(* Verify that the statuses of the switchbox pumps match the expected statuses *)
FUNCTION F_VerifySBPumpStatuses : BOOL
VAR_INPUT
	stExpStatus : ST_SBPumpStatuses; // The expected state of the system
	bEnforce : BOOL; // Whether to try forcing the states
END_VAR
VAR
	stStatus : ST_SBPumpStatuses;
END_VAR

stStatus := F_GetSBPumpStatuses();

IF bEnforce THEN
	// Try setting system states to the expected states
	F_SetSBPumpStatuses(stExpStatus);
END_IF

// Return true if the expected status matches the actual status
F_VerifySBPumpStatuses := stExpStatus.bRoughingPumpOn = stStatus.bRoughingPumpOn
	AND stExpStatus.bTurboPumpOn = stStatus.bTurboPumpOn
	AND stExpStatus.bIonPumpOn = stStatus.bIonPumpOn;

END_FUNCTION

(* stored: Version 1.1.0.1, ProductVersion 3.1.4022.17
   POU F_VerifySBPumpStatuses: Id {f4b16073-0e15-47a9-978a-2d5792f30146}, SpecialFunc None *)
